(*			
	RAFALOS
	Rafał Osajda		19.09.2025		TC 4024.66
	Element bazowy umożliwiający potomkom wysyłaś zgłoszenia do logera
*)
FUNCTION_BLOCK FB_LoggerElement 
VAR
	itfLogger				: ITF_Logger;
	
END_VAR

END_FUNCTION_BLOCK

(* stored: Version 1.1.0.1
   POU FB_LoggerElement: Id {84ce134f-38cc-08bd-3d60-40e507799b32}, SpecialFunc None *)
